FUNCTION_BLOCK Sensors (* Composite Function Block Type *)
  (* Standard: 61499-2 *)
  (* Version 1.0, 2019-05-09, jetbrains *)
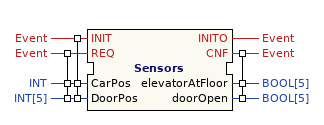
  EVENT_INPUT
    INIT WITH CarPos, DoorPos; (* Initialization Request *)
    REQ WITH CarPos, DoorPos; (* Normal Execution Request *)
  END_EVENT
  EVENT_OUTPUT
    INITO; (* Initialization Confirm *)
    CNF WITH elevatorAtFloor, doorOpen; (* Execution Confirmation *)
  END_EVENT
  VAR_INPUT
    CarPos : INT; (* Input event qualifier *)
    DoorPos : ARRAY [0..4] OF INT;
  END_VAR
  VAR_OUTPUT
    elevatorAtFloor : ARRAY [0..4] OF BOOL; (* Output event qualifier *)
    doorOpen : ARRAY [0..4] OF BOOL;
  END_VAR
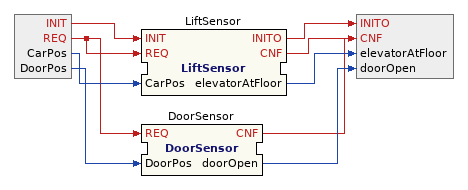
  FBS
    LiftSensor : LiftSensor;
    DoorSensor : DoorSensor;
  END_FBS
  EVENT_CONNECTIONS
    REQ TO LiftSensor.REQ;
    LiftSensor.CNF TO CNF;
    REQ TO DoorSensor.REQ;
    DoorSensor.CNF TO CNF;
    INIT TO LiftSensor.INIT;
    LiftSensor.INITO TO INITO;
  END_CONNECTIONS
  DATA_CONNECTIONS
    CarPos TO LiftSensor.CarPos;
    DoorPos TO DoorSensor.DoorPos;
    DoorSensor.doorOpen TO doorOpen;
    LiftSensor.elevatorAtFloor TO elevatorAtFloor;
  END_CONNECTIONS
END_FUNCTION_BLOCK
